TYPE ST_AKM_Zustand :
STRUCT
	Temp_HW_Vorl		: REAL;
	Temp_HW_Rueckl	: REAL;
	Temp_WW_Vorl		: REAL;
	Temp_WW_Rueckl	: REAL;
	Temp_KW_Vorl		: REAL;
	Temp_KW_Rueckl	: REAL;

	Anforderung_Kaelte	: BOOL; (* Wert wird über OPCUA geschrieben *)
	Anforderung_Warme	: BOOL;	(* Wert wird über OPCUA geschrieben *)
	Betrieb_REAL				: REAL;
	Freigabe				: BOOL;
	Freigabe_Deakt		: BOOL;
	Freigabe_Code		: WORD;

	Kommunikation		: BOOL;

	Stoerung			: BOOL;
	Stoerung_Code		: WORD;
	Vorlauf_Nachlauf	: BOOL; (*wird von OPCUA ausgelesen*)
	Warnung				: BOOL;
	Warnung_Code		: WORD;
END_STRUCT
END_TYPE

(* stored: Version 1.1.0.1, ProductVersion 3.1.4024.9
   DUT ST_AKM_Zustand: Id {60600fb0-8820-4fa5-b203-ea83b56daf91} *)
